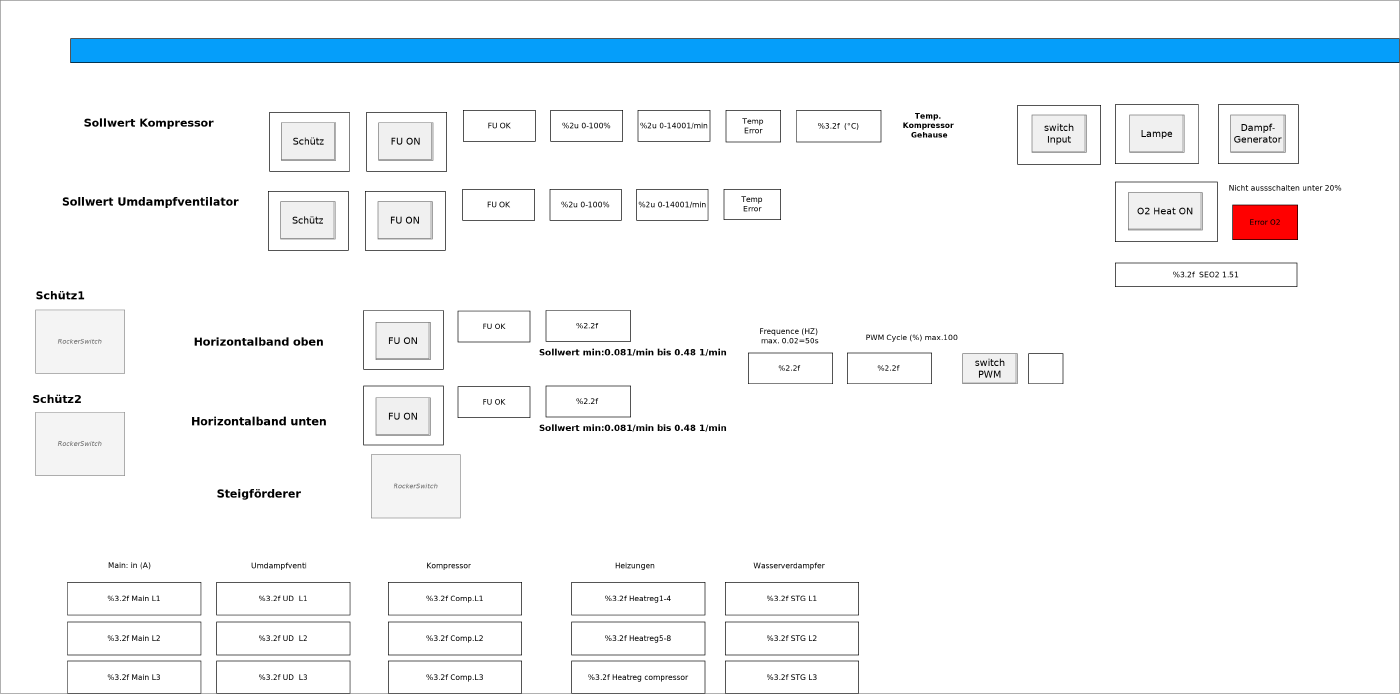
VISUALIZATION Main  // 2147x1065, background image backround
    Rectangle (1560,161 128x91), colour toggle: switch_Setpoint_Value
    Rectangle (108,59 2039x37)
    Rectangle (844,169 111x48), "%2u 0-100%", tooltip "Durchmesser in mm eingeben", text variable: GVL.Setpoint_Compressor_Visu
        OnMouseDown: write the text variable via VisuDialogs.Numpad, min 0, max 100
    Rectangle (837,592 130x48), "%2.2f", text variable: Setpoint_Belts_Visu_bottom_1_min
        OnMouseDown: write the text variable via VisuDialogs.Numpad, min 0.0, max 0.48
    Rectangle (1113,169 84x49), "Temp Error", colour toggle: GVL.Compressor_PT100_error
    Rectangle (843,290 110x48), "%2u 0-100%", tooltip "Durchmesser in mm eingeben", text variable: GVL.Setpoint_SteamFan_Visu
        OnMouseDown: write the text variable via VisuDialogs.Numpad, min 0, max 100
    Rectangle (1110,290 87x47), "Temp Error"
    Rectangle (1221,169 130x49), "%3.2f (°C)", tooltip "Durchmesser in mm eingeben", text variable: GVL.T_Ueberwachung_scroll_comp
    Rectangle (1339,161 173x63), "Temp. Kompressor Gehause"
    Textfield (84,172 288x33), "Sollwert Kompressor"
    Textfield (84,293 293x33), "Sollwert Umdampfventilator"
    Textfield (253,630 288x33), "Horizontalband unten"
    Textfield (253,741 288x33), "Steigförderer"
    Rectangle (411,293 123x91), colour toggle: GVL.SteamFAN_Switch_ON_manu
    Button (430,309 84x58), "Schütz", pressed state: GVL.SteamFAN_Switch_ON_manu
        toggle GVL.SteamFAN_Switch_ON_manu
    Rectangle (413,172 123x91), colour toggle: GVL.Compressor_Switch_ON_Manu
    Button (431,188 84x58), "Schütz", pressed state: GVL.Compressor_Switch_ON_Manu
        toggle GVL.Compressor_Switch_ON_Manu
    Rectangle (562,172 123x91), colour toggle: GVL.Compressor_ON_Manu
    Button (580,188 84x58), "FU ON", pressed state: GVL.Compressor_ON_Manu
        toggle GVL.Compressor_ON_Manu
    Rectangle (710,169 111x48), "FU OK", colour toggle: GVL.Compressor_OK
    Rectangle (709,290 111x48), "FU OK", colour toggle: GVL.SteamFan_OK
    Rectangle (557,592 123x91), colour toggle: GVL.Belts_ON_bottom_Manu
    Button (576,610 84x58), "FU ON", pressed state: GVL.Belts_ON_bottom_Manu
        toggle GVL.Belts_ON_bottom_Manu
    Rectangle (702,593 111x48), "FU OK", colour toggle: GVL.Belts_bottom_OK
    Rectangle (560,293 123x91), colour toggle: GVL.SteamFan_ON_manu
    Button (579,309 84x58), "FU ON"
        toggle GVL.SteamFan_ON_manu
    Rectangle (332,893 205x51), "%3.2f UD L1", tooltip "Durchmesser in mm eingeben", text variable: Current_OUT_Fan_L1
    Rectangle (332,954 205x51), "%3.2f UD L2", tooltip "Durchmesser in mm eingeben", text variable: Current_OUT_Fan_L2
    Rectangle (332,1014 205x51), "%3.2f UD L3", tooltip "Durchmesser in mm eingeben", text variable: Current_OUT_Fan_L3
    Rectangle (876,893 205x51), "%3.2f Heatreg1-4", tooltip "Durchmesser in mm eingeben", text variable: Current_OUT_Heatreg_1_TO_4
    Rectangle (876,954 205x51), "%3.2f Heatreg5-8", tooltip "Durchmesser in mm eingeben", text variable: Current_OUT_Heatreg_5_TO_8
    Rectangle (876,1014 205x51), "%3.2f Heatreg compressor", tooltip "Durchmesser in mm eingeben", text variable: Current_OUT_Heatreg_Compressor
    Rectangle (123,849 151x37), "Main: in (A)"
    Rectangle (103,893 205x51), "%3.2f Main L1", tooltip "Durchmesser in mm eingeben", text variable: GVL.Current_OUT_Complete_L1
    Rectangle (103,954 205x51), "%3.2f Main L2", tooltip "Durchmesser in mm eingeben", text variable: GVL.Current_OUT_Complete_L2
    Rectangle (103,1014 205x51), "%3.2f Main L3", tooltip "Durchmesser in mm eingeben", text variable: GVL.Current_OUT_Complete_L3
    Rectangle (595,893 205x51), "%3.2f Comp.L1", tooltip "Durchmesser in mm eingeben", text variable: GVL.Current_OUT_Compressor_L1
    Rectangle (595,954 205x51), "%3.2f Comp.L2", tooltip "Durchmesser in mm eingeben", text variable: GVL.Current_OUT_Compressor_L2
    Rectangle (595,1014 205x51), "%3.2f Comp.L3", tooltip "Durchmesser in mm eingeben", text variable: GVL.Current_OUT_Compressor_L3
    Rectangle (582,857 212x22), "Kompressor"
    Rectangle (849,857 250x22), "Heizungen"
    Rectangle (322,857 212x22), "Umdampfventi"
    Rectangle (1112,893 205x51), "%3.2f STG L1", tooltip "Durchmesser in mm eingeben", text variable: Current_OUT_SteamGen1
    Rectangle (1112,954 205x51), "%3.2f STG L2", tooltip "Durchmesser in mm eingeben", text variable: Current_OUT_SteamGen2
    Rectangle (1112,1014 205x51), "%3.2f STG L3", tooltip "Durchmesser in mm eingeben", text variable: Current_OUT_SteamGen3
    Rectangle (1085,857 250x22), "Wasserverdampfer"
    Rectangle (1710,160 128x91), colour toggle: MAIN_ON_Switch_Light_visu
    Button (1732,176 84x58), "Lampe", pressed state: GVL.Belts_TOP_Switch_ON_Manu, input disabled if: GVL.Control_Manu_active=False
        toggle MAIN_ON_Switch_Light_visu
    Rectangle (1868,160 123x91), colour toggle: MAIN_ON_STEAM_GEN
    Button (1887,176 84x58), "Dampf- Generator", pressed state: GVL.Belts_TOP_Switch_ON_Manu, input disabled if: GVL.Control_Manu_active=FALSE
        toggle MAIN_ON_STEAM_GEN
    Textfield (805,642 331x30), "Sollwert min:0.081/min bis 0.48 1/min"
    Rectangle (1710,403 279x37), "%3.2f SEO2 1.51", tooltip "Durchmesser in mm eingeben", text variable: GVL.O2_Visu
    Rectangle (1710,279 157x92), colour toggle: O2_Sensor_Start
    Button (1730,295 114x58), "O2 Heat ON", pressed state: GVL.Belts_TOP_Switch_ON_Manu, input disabled if: DO_not_turn_off_Heating_O2_Sensor
        toggle O2_Sensor_Start
    Rectangle (1890,314 100x54), "Error O2", colour toggle: O2_Sensor_Error
    Rectangle (1862,270 218x37), "Nicht aussschalten unter 20%"
    Rectangle (978,169 111x48), "%2u 0-14001/min", tooltip "Durchmesser in mm eingeben", text variable: Setpoint_1_MIN_Compressor_IN
        OnMouseDown: write the text variable via VisuDialogs.Numpad, min 0, max 100
    Rectangle (976,290 110x48), "%2u 0-14001/min", tooltip "Durchmesser in mm eingeben", text variable: GVL.Setpoint_SteamFan_Visu
        OnMouseDown: write the text variable via VisuDialogs.Numpad, min 0, max 100
    Button (1582,176 84x58), "switch Input", pressed state: GVL.Belts_TOP_Switch_ON_Manu
        toggle switch_Setpoint_Value p2164770859=TRUE
    Rectangle (837,476 130x48), "%2.2f", text variable: Setpoint_Belts_Visu_TOP_1_min
        OnMouseDown: write the text variable via VisuDialogs.Numpad, min 0.0, max 0.48
    Textfield (253,508 288x33), "Horizontalband oben"
    Rectangle (557,476 123x91), colour toggle: GVL.Belts_ON_TOP_Manu
    Button (576,494 84x58), "FU ON", pressed state: GVL.Belts_ON_TOP_Manu
        toggle GVL.Belts_ON_TOP_Manu
    Rectangle (702,477 111x48), "FU OK", colour toggle: GVL.Belts_OK_TOP
    Textfield (805,526 331x30), "Sollwert min:0.081/min bis 0.48 1/min"
    Rectangle (1147,541 130x48), "%2.2f", text variable: Base_Frequence_Main_Belt
        OnMouseDown: write the text variable via VisuDialogs.Numpad, min 0, max 10
    Rectangle (1299,541 130x48), "%2.2f", text variable: Main_Belt_PWMDutyCycle_VISU
        OnMouseDown: write the text variable via VisuDialogs.Numpad, min 20, max 100
    Rectangle (1143,496 137x40), "Frequence (HZ) max. 0.02=50s"
    Rectangle (1304,507 189x22), "PWM Cycle (%) max.100"
    Rectangle (1577,542 53x47), colour toggle: Switch_ON_Main_Belt_PWM
    Button (1476,542 84x47), "switch PWM", pressed state: GVL.Belts_TOP_Switch_ON_Manu
        toggle Switch_ON_Main_Belt_PWM p2164770859=TRUE
    RockerSwitch (54,475 137x98), variable: Circuit_1_ON, behaviour: TOGGLE, style: Switch-RockerSwitch-Gray
    RockerSwitch (54,632 137x98), variable: Circuit_2_ON, behaviour: TOGGLE, style: Switch-RockerSwitch-Gray
    RockerSwitch (569,697 137x98), variable: GVL.M_Belt_Feeder_ON_Manu, behaviour: TOGGLE, style: Switch-RockerSwitch-Gray
    Textfield (29,437 127x33), "Schütz1"
    Textfield (24,596 127x33), "Schütz2"
END_VISUALIZATION

(* stored: Version 1.1.0.1, ProductVersion 3.1.4024.3
   Visu Main: Id {bd6a4bd9-71fe-4460-97b9-2bcfb92de9b6} *)
